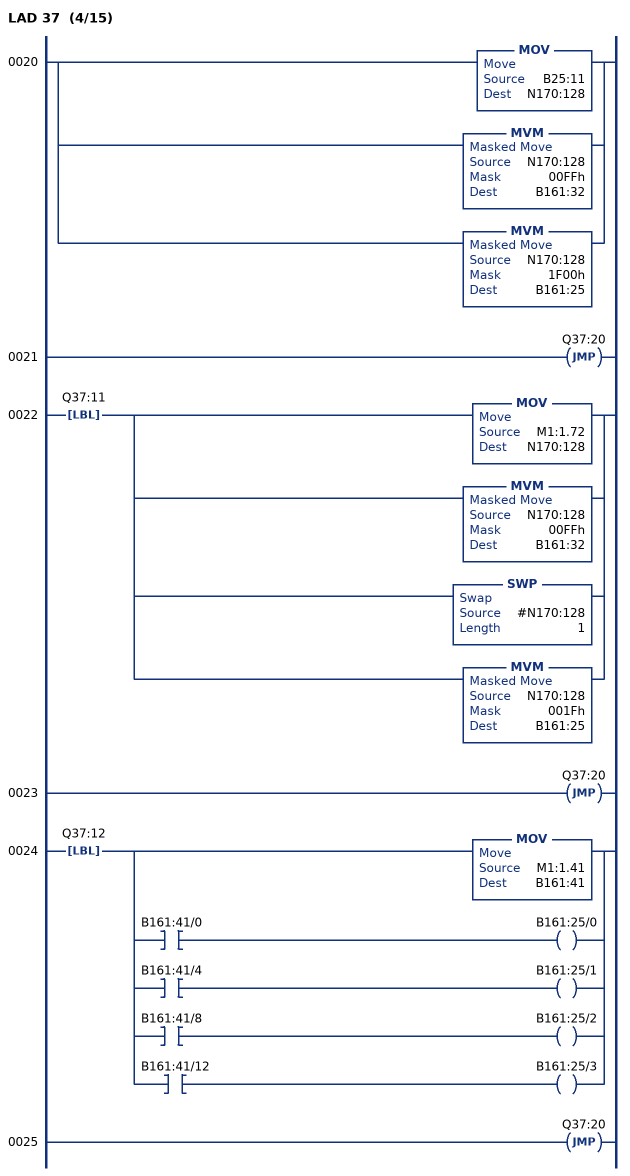
% Rung: 20 %
SOR BST MOV B25:11 N170:128 NXB MVM N170:128 00FFh B161:32 NXB MVM N170:128 1F00h B161:25 BND EOR
% Rung: 21 %
SOR JMP Q37:20 EOR
% Rung: 22 %
SOR LBL Q37:11 BST MOV M1:1.72 N170:128 NXB MVM N170:128 00FFh B161:32 NXB SWP #N170:128 1 NXB MVM N170:128 001Fh B161:25 BND EOR
% Rung: 23 %
SOR JMP Q37:20 EOR
% Rung: 24 %
SOR LBL Q37:12 BST MOV M1:1.41 B161:41 NXB XIC B161:41/0 OTE B161:25/0 NXB XIC B161:41/4 OTE B161:25/1 NXB XIC B161:41/8 OTE B161:25/2 NXB XIC B161:41/12 OTE B161:25/3 BND EOR
% Rung: 25 %
SOR JMP Q37:20 EOR

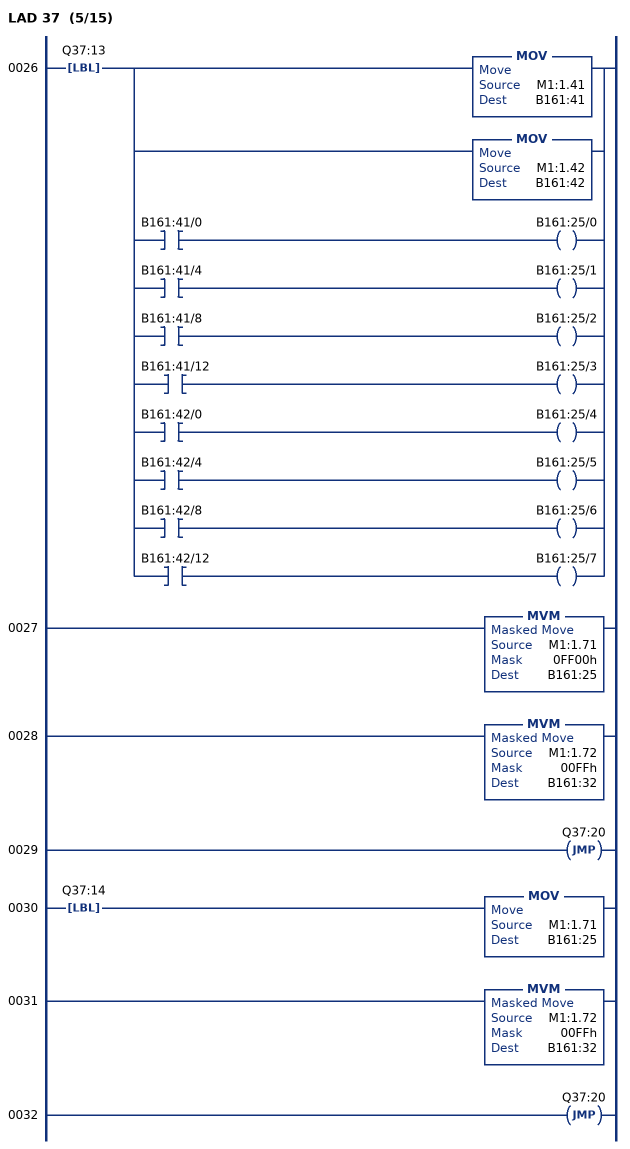
% Rung: 26 %
SOR LBL Q37:13 BST MOV M1:1.41 B161:41 NXB MOV M1:1.42 B161:42 NXB XIC B161:41/0 OTE B161:25/0 NXB XIC B161:41/4 OTE B161:25/1 NXB XIC B161:41/8 OTE B161:25/2 NXB XIC B161:41/12 OTE B161:25/3 NXB XIC B161:42/0 OTE B161:25/4 NXB XIC B161:42/4 OTE B161:25/5 NXB XIC B161:42/8 OTE B161:25/6 NXB XIC B161:42/12 OTE B161:25/7 BND EOR
% Rung: 27 %
SOR MVM M1:1.71 0FF00h B161:25 EOR
% Rung: 28 %
SOR MVM M1:1.72 00FFh B161:32 EOR
% Rung: 29 %
SOR JMP Q37:20 EOR
% Rung: 30 %
SOR LBL Q37:14 MOV M1:1.71 B161:25 EOR
% Rung: 31 %
SOR MVM M1:1.72 00FFh B161:32 EOR
% Rung: 32 %
SOR JMP Q37:20 EOR

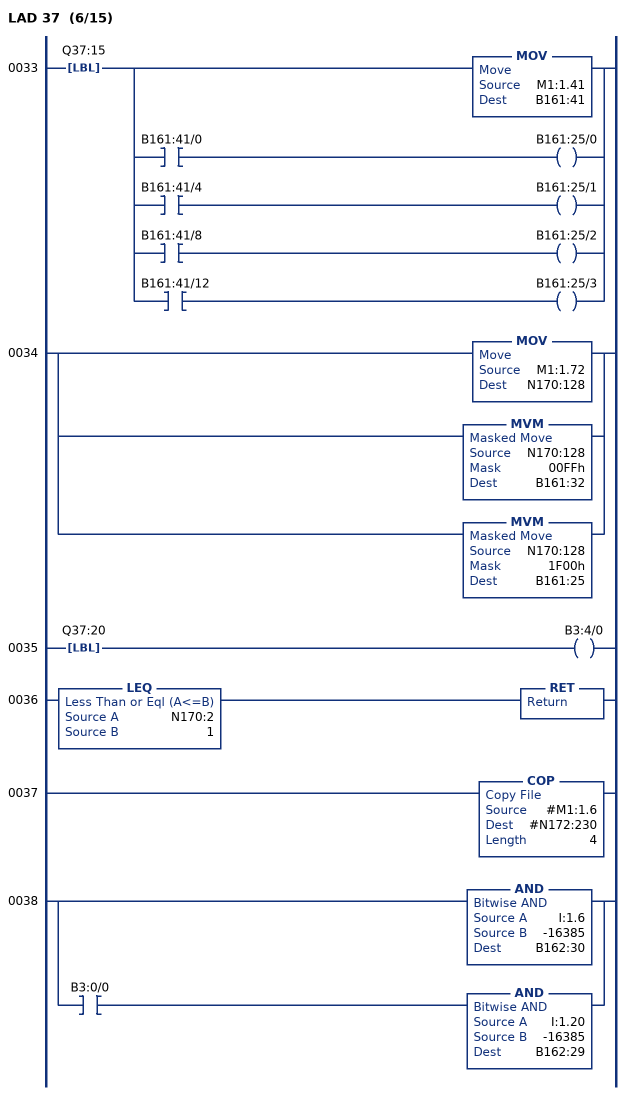
% Rung: 33 %
SOR LBL Q37:15 BST MOV M1:1.41 B161:41 NXB XIC B161:41/0 OTE B161:25/0 NXB XIC B161:41/4 OTE B161:25/1 NXB XIC B161:41/8 OTE B161:25/2 NXB XIC B161:41/12 OTE B161:25/3 BND EOR
% Rung: 34 %
SOR BST MOV M1:1.72 N170:128 NXB MVM N170:128 00FFh B161:32 NXB MVM N170:128 1F00h B161:25 BND EOR
% Rung: 35 %
SOR LBL Q37:20 OTE B3:4/0 EOR
% Rung: 36 %
SOR LEQ N170:2 1 RET EOR
% Rung: 37 %
SOR COP #M1:1.6 #N172:230 4 EOR
% Rung: 38 %
SOR BST AND I:1.6 -16385 B162:30 NXB XIC B3:0/0 AND I:1.20 -16385 B162:29 BND EOR

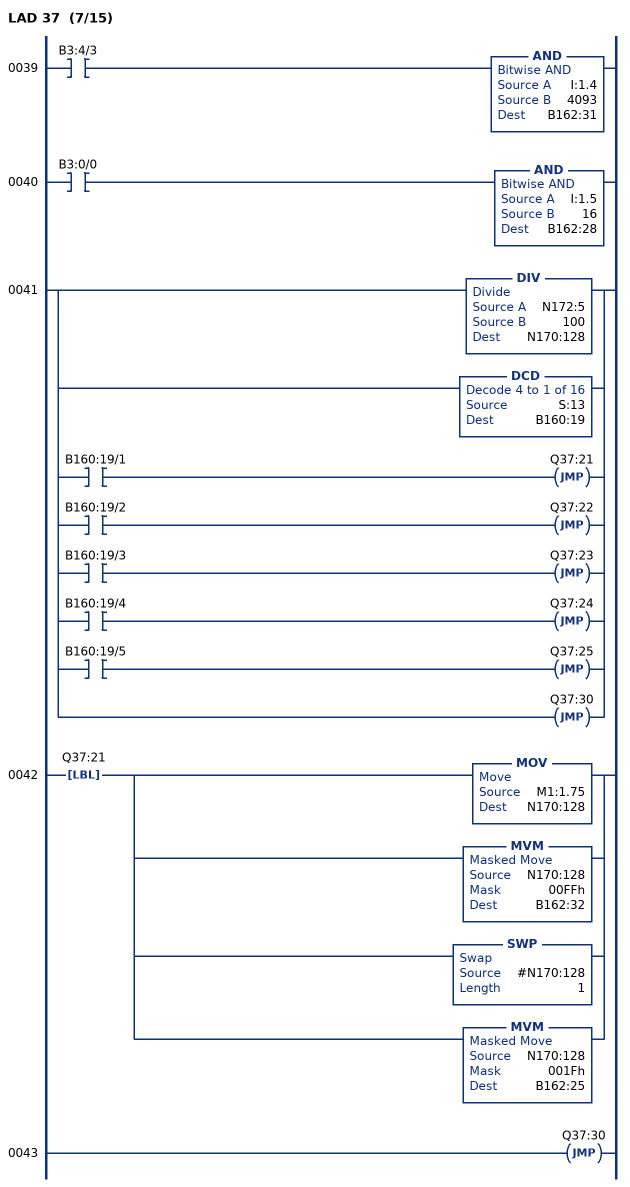
% Rung: 39 %
SOR XIC B3:4/3 AND I:1.4 4093 B162:31 EOR
% Rung: 40 %
SOR XIC B3:0/0 AND I:1.5 16 B162:28 EOR
% Rung: 41 %
SOR BST DIV N172:5 100 N170:128 NXB DCD S:13 B160:19 NXB BST XIC B160:19/1 JMP Q37:21 NXB XIC B160:19/2 JMP Q37:22 NXB XIC B160:19/3 JMP Q37:23 NXB XIC B160:19/4 JMP Q37:24 NXB XIC B160:19/5 JMP Q37:25 BND NXB JMP Q37:30 BND EOR
%   S:13  "Math Register" %
% Rung: 42 %
SOR LBL Q37:21 BST MOV M1:1.75 N170:128 NXB MVM N170:128 00FFh B162:32 NXB SWP #N170:128 1 NXB MVM N170:128 001Fh B162:25 BND EOR
% Rung: 43 %
SOR JMP Q37:30 EOR

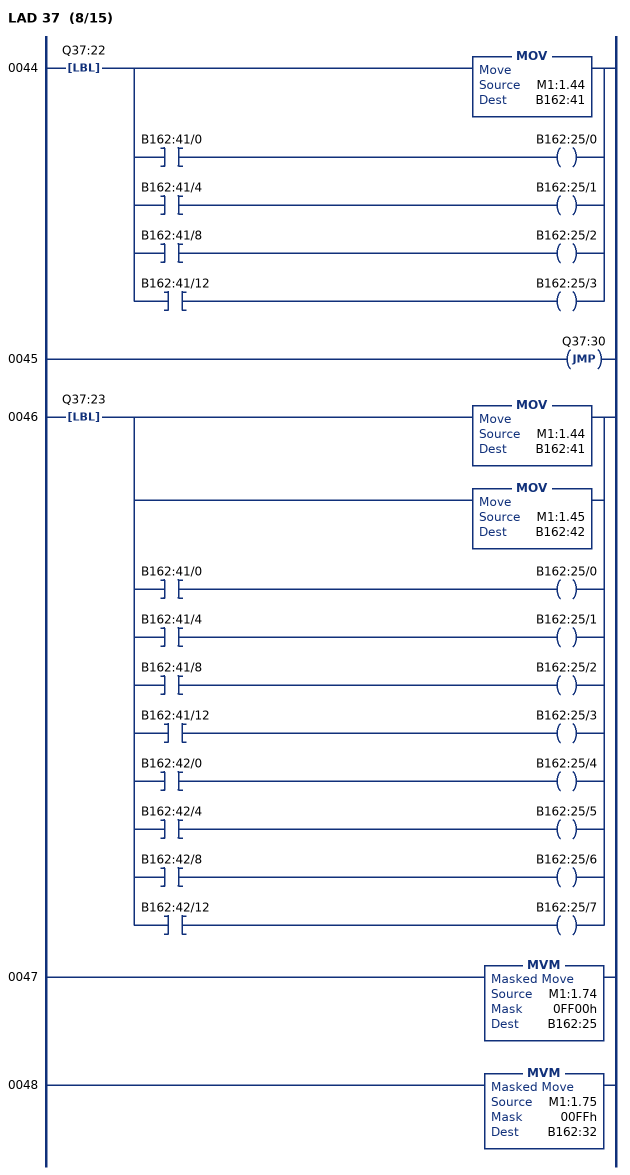
% Rung: 44 %
SOR LBL Q37:22 BST MOV M1:1.44 B162:41 NXB XIC B162:41/0 OTE B162:25/0 NXB XIC B162:41/4 OTE B162:25/1 NXB XIC B162:41/8 OTE B162:25/2 NXB XIC B162:41/12 OTE B162:25/3 BND EOR
% Rung: 45 %
SOR JMP Q37:30 EOR
% Rung: 46 %
SOR LBL Q37:23 BST MOV M1:1.44 B162:41 NXB MOV M1:1.45 B162:42 NXB XIC B162:41/0 OTE B162:25/0 NXB XIC B162:41/4 OTE B162:25/1 NXB XIC B162:41/8 OTE B162:25/2 NXB XIC B162:41/12 OTE B162:25/3 NXB XIC B162:42/0 OTE B162:25/4 NXB XIC B162:42/4 OTE B162:25/5 NXB XIC B162:42/8 OTE B162:25/6 NXB XIC B162:42/12 OTE B162:25/7 BND EOR
% Rung: 47 %
SOR MVM M1:1.74 0FF00h B162:25 EOR
% Rung: 48 %
SOR MVM M1:1.75 00FFh B162:32 EOR

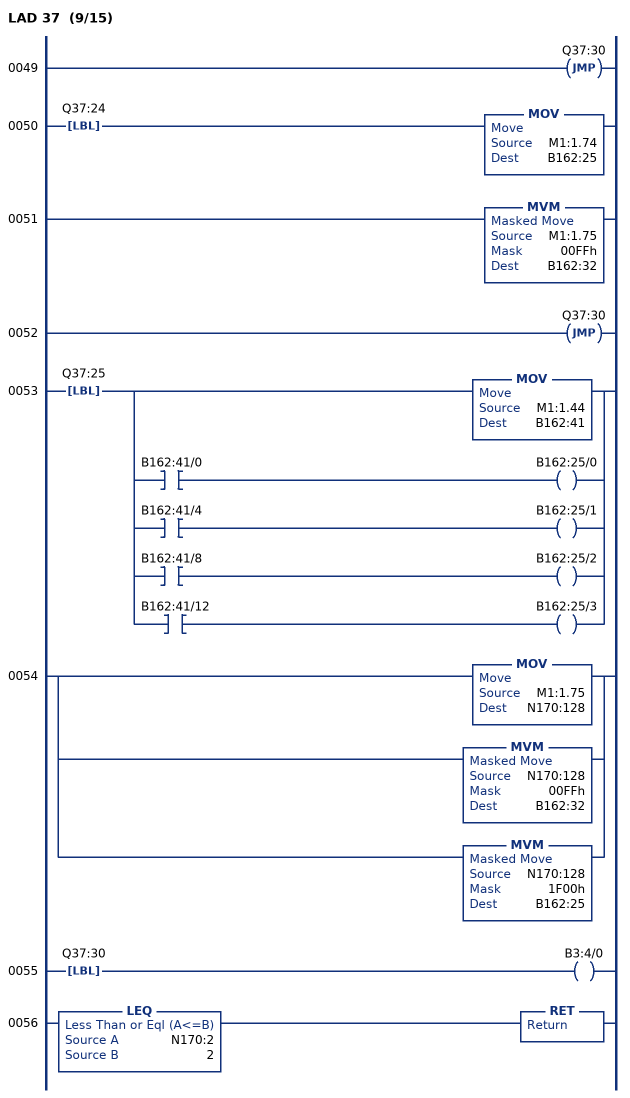
% Rung: 49 %
SOR JMP Q37:30 EOR
% Rung: 50 %
SOR LBL Q37:24 MOV M1:1.74 B162:25 EOR
% Rung: 51 %
SOR MVM M1:1.75 00FFh B162:32 EOR
% Rung: 52 %
SOR JMP Q37:30 EOR
% Rung: 53 %
SOR LBL Q37:25 BST MOV M1:1.44 B162:41 NXB XIC B162:41/0 OTE B162:25/0 NXB XIC B162:41/4 OTE B162:25/1 NXB XIC B162:41/8 OTE B162:25/2 NXB XIC B162:41/12 OTE B162:25/3 BND EOR
% Rung: 54 %
SOR BST MOV M1:1.75 N170:128 NXB MVM N170:128 00FFh B162:32 NXB MVM N170:128 1F00h B162:25 BND EOR
% Rung: 55 %
SOR LBL Q37:30 OTE B3:4/0 EOR
% Rung: 56 %
SOR LEQ N170:2 2 RET EOR

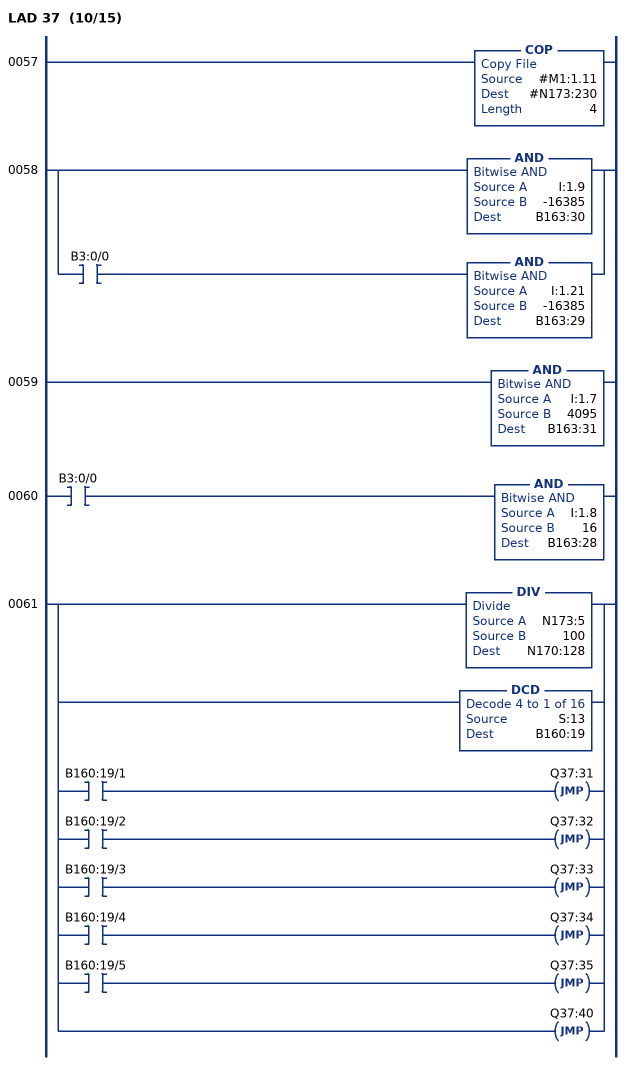
% Rung: 57 %
SOR COP #M1:1.11 #N173:230 4 EOR
% Rung: 58 %
SOR BST AND I:1.9 -16385 B163:30 NXB XIC B3:0/0 AND I:1.21 -16385 B163:29 BND EOR
% Rung: 59 %
SOR AND I:1.7 4095 B163:31 EOR
% Rung: 60 %
SOR XIC B3:0/0 AND I:1.8 16 B163:28 EOR
% Rung: 61 %
SOR BST DIV N173:5 100 N170:128 NXB DCD S:13 B160:19 NXB BST XIC B160:19/1 JMP Q37:31 NXB XIC B160:19/2 JMP Q37:32 NXB XIC B160:19/3 JMP Q37:33 NXB XIC B160:19/4 JMP Q37:34 NXB XIC B160:19/5 JMP Q37:35 BND NXB JMP Q37:40 BND EOR
%   S:13  "Math Register" %

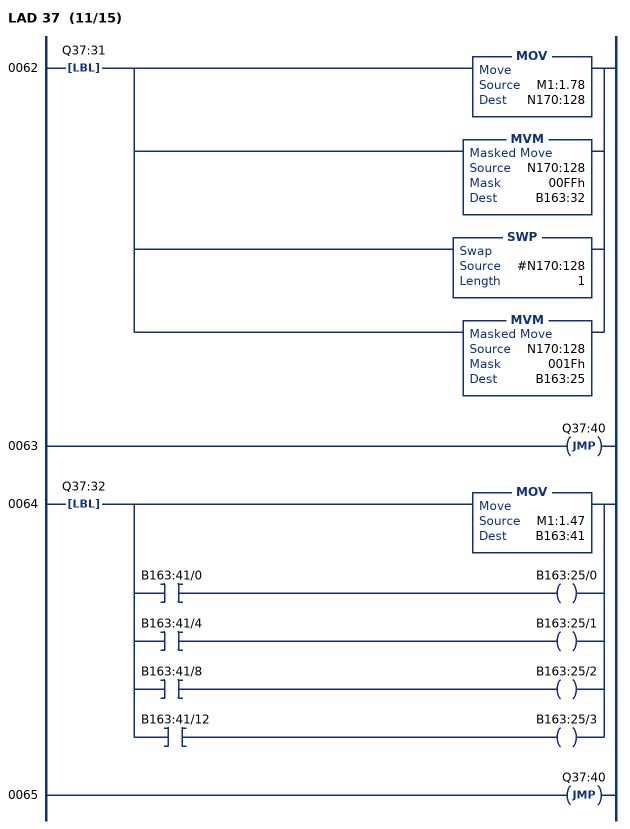
% Rung: 62 %
SOR LBL Q37:31 BST MOV M1:1.78 N170:128 NXB MVM N170:128 00FFh B163:32 NXB SWP #N170:128 1 NXB MVM N170:128 001Fh B163:25 BND EOR
% Rung: 63 %
SOR JMP Q37:40 EOR
% Rung: 64 %
SOR LBL Q37:32 BST MOV M1:1.47 B163:41 NXB XIC B163:41/0 OTE B163:25/0 NXB XIC B163:41/4 OTE B163:25/1 NXB XIC B163:41/8 OTE B163:25/2 NXB XIC B163:41/12 OTE B163:25/3 BND EOR
% Rung: 65 %
SOR JMP Q37:40 EOR

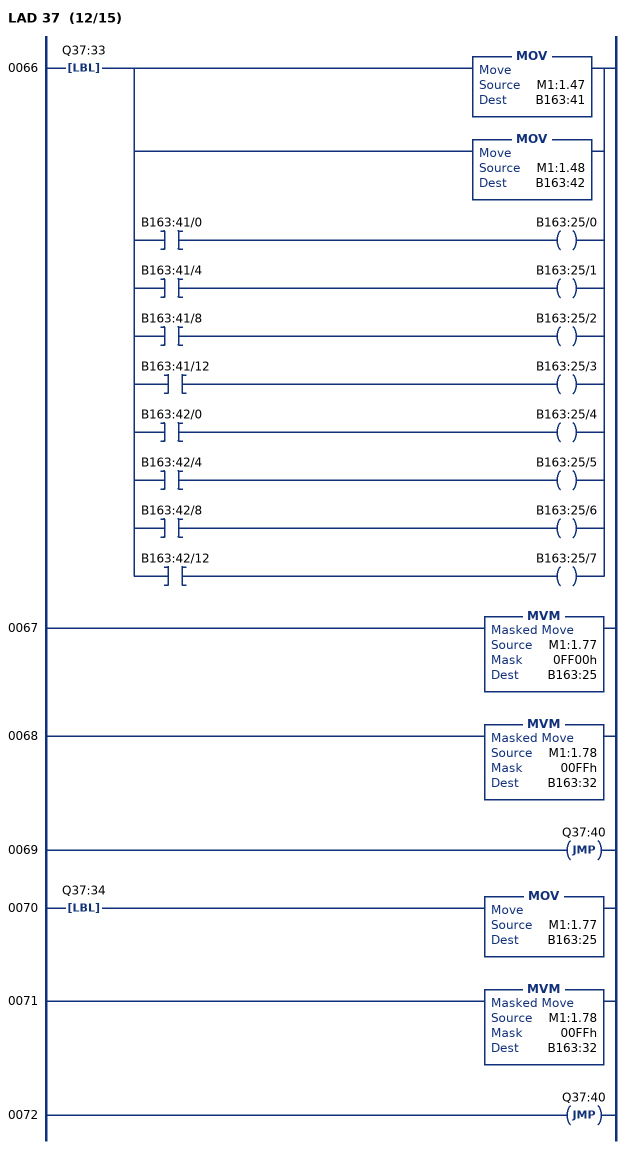
% Rung: 66 %
SOR LBL Q37:33 BST MOV M1:1.47 B163:41 NXB MOV M1:1.48 B163:42 NXB XIC B163:41/0 OTE B163:25/0 NXB XIC B163:41/4 OTE B163:25/1 NXB XIC B163:41/8 OTE B163:25/2 NXB XIC B163:41/12 OTE B163:25/3 NXB XIC B163:42/0 OTE B163:25/4 NXB XIC B163:42/4 OTE B163:25/5 NXB XIC B163:42/8 OTE B163:25/6 NXB XIC B163:42/12 OTE B163:25/7 BND EOR
% Rung: 67 %
SOR MVM M1:1.77 0FF00h B163:25 EOR
% Rung: 68 %
SOR MVM M1:1.78 00FFh B163:32 EOR
% Rung: 69 %
SOR JMP Q37:40 EOR
% Rung: 70 %
SOR LBL Q37:34 MOV M1:1.77 B163:25 EOR
% Rung: 71 %
SOR MVM M1:1.78 00FFh B163:32 EOR
% Rung: 72 %
SOR JMP Q37:40 EOR

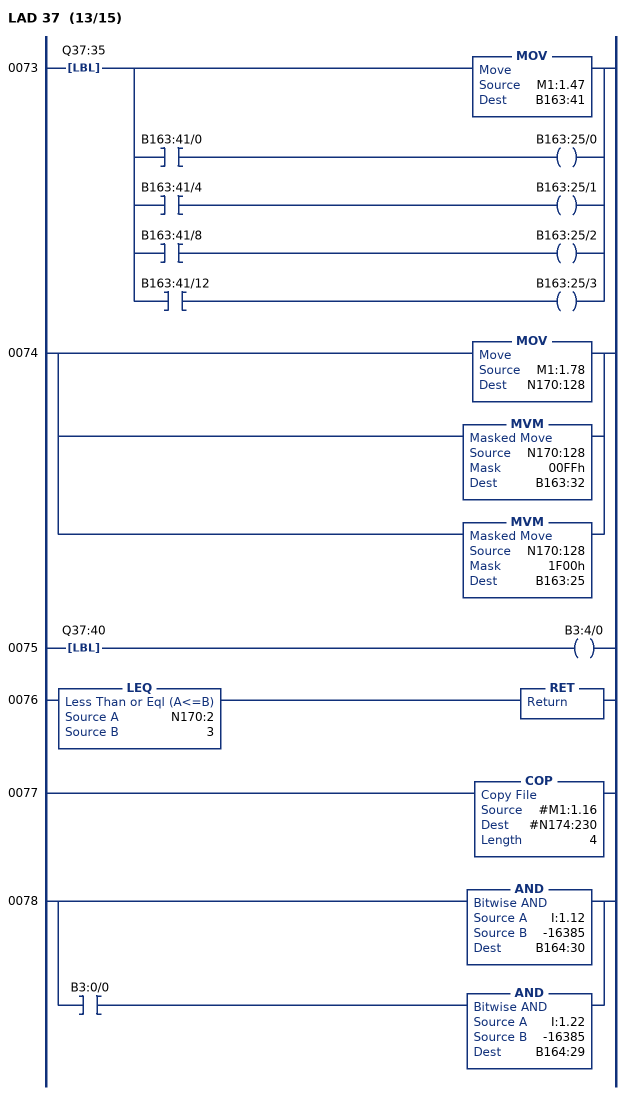
% Rung: 73 %
SOR LBL Q37:35 BST MOV M1:1.47 B163:41 NXB XIC B163:41/0 OTE B163:25/0 NXB XIC B163:41/4 OTE B163:25/1 NXB XIC B163:41/8 OTE B163:25/2 NXB XIC B163:41/12 OTE B163:25/3 BND EOR
% Rung: 74 %
SOR BST MOV M1:1.78 N170:128 NXB MVM N170:128 00FFh B163:32 NXB MVM N170:128 1F00h B163:25 BND EOR
% Rung: 75 %
SOR LBL Q37:40 OTE B3:4/0 EOR
% Rung: 76 %
SOR LEQ N170:2 3 RET EOR
% Rung: 77 %
SOR COP #M1:1.16 #N174:230 4 EOR
% Rung: 78 %
SOR BST AND I:1.12 -16385 B164:30 NXB XIC B3:0/0 AND I:1.22 -16385 B164:29 BND EOR

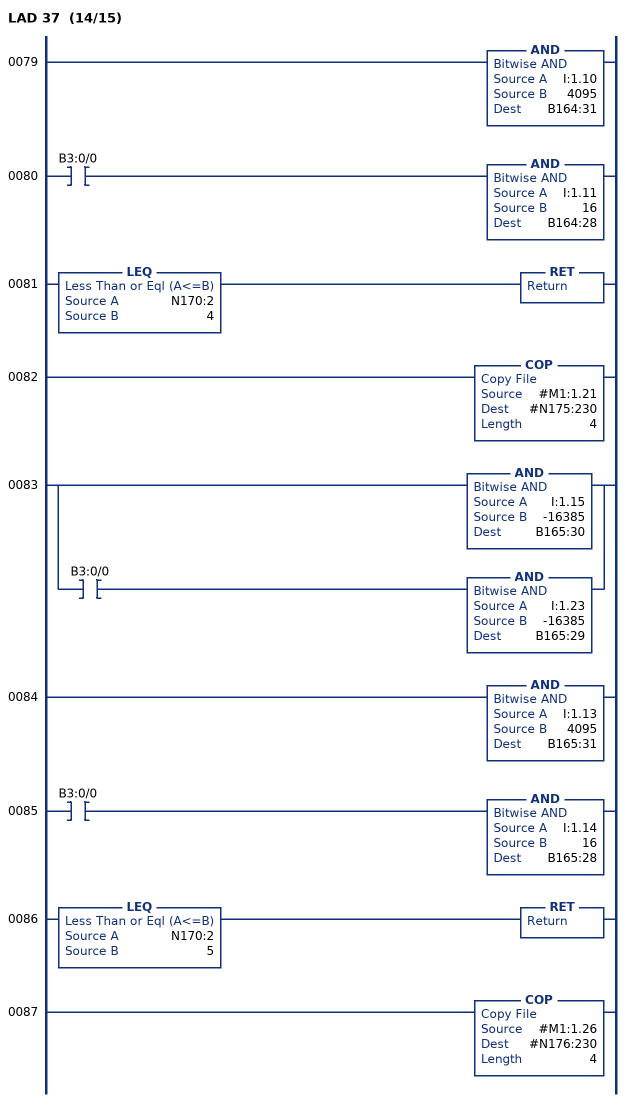
% Rung: 79 %
SOR AND I:1.10 4095 B164:31 EOR
% Rung: 80 %
SOR XIC B3:0/0 AND I:1.11 16 B164:28 EOR
% Rung: 81 %
SOR LEQ N170:2 4 RET EOR
% Rung: 82 %
SOR COP #M1:1.21 #N175:230 4 EOR
% Rung: 83 %
SOR BST AND I:1.15 -16385 B165:30 NXB XIC B3:0/0 AND I:1.23 -16385 B165:29 BND EOR
% Rung: 84 %
SOR AND I:1.13 4095 B165:31 EOR
% Rung: 85 %
SOR XIC B3:0/0 AND I:1.14 16 B165:28 EOR
% Rung: 86 %
SOR LEQ N170:2 5 RET EOR
% Rung: 87 %
SOR COP #M1:1.26 #N176:230 4 EOR

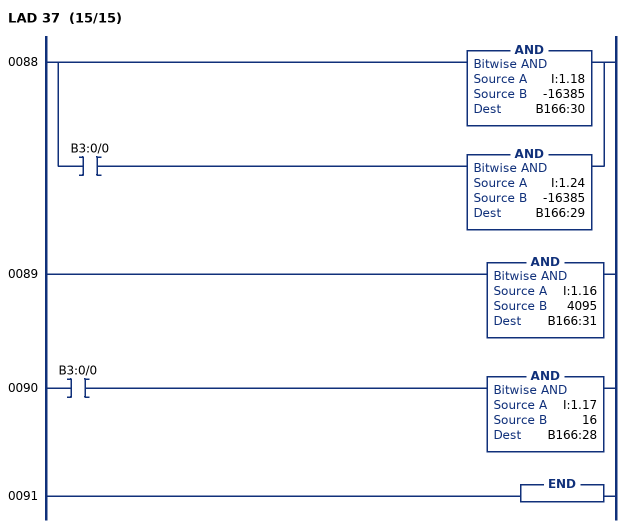
% Rung: 88 %
SOR BST AND I:1.18 -16385 B166:30 NXB XIC B3:0/0 AND I:1.24 -16385 B166:29 BND EOR
% Rung: 89 %
SOR AND I:1.16 4095 B166:31 EOR
% Rung: 90 %
SOR XIC B3:0/0 AND I:1.17 16 B166:28 EOR
% Rung: 91 %
SOR END EOR

LADDER 38
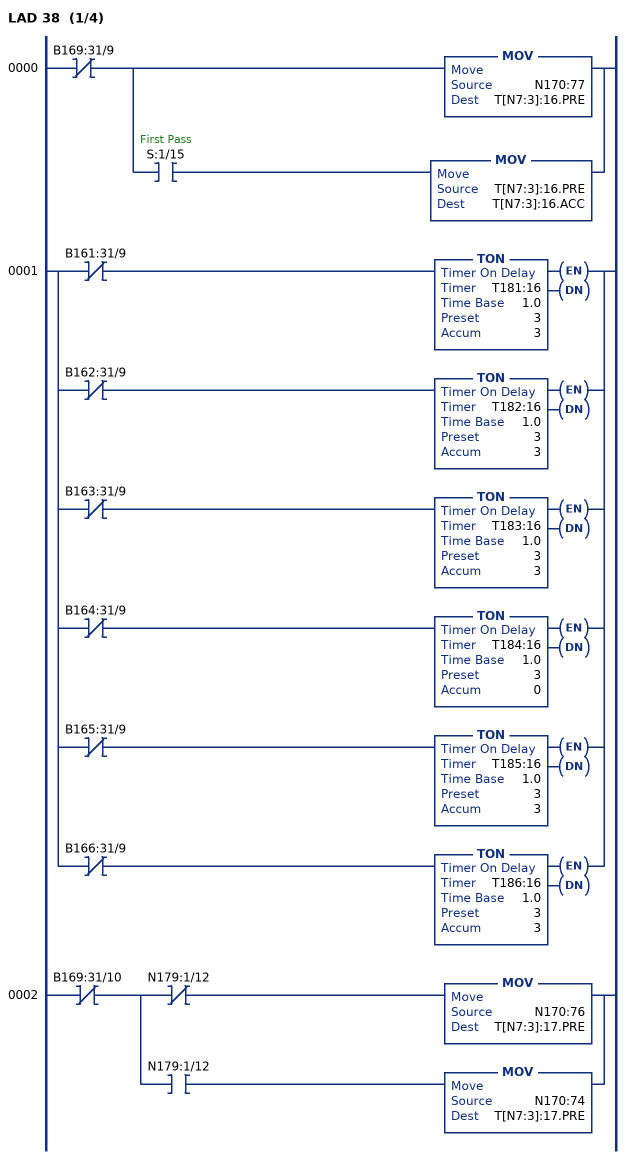
% Rung: 0 %
SOR XIO B169:31/9 BST MOV N170:77 T[N7:3]:16.PRE NXB XIC S:1/15 MOV T[N7:3]:16.PRE T[N7:3]:16.ACC BND EOR
%   S:1/15  "First Pass" %
% Rung: 1 %
SOR BST XIO B161:31/9 TON T181:16 1.0 3 3 NXB XIO B162:31/9 TON T182:16 1.0 3 3 NXB XIO B163:31/9 TON T183:16 1.0 3 3 NXB XIO B164:31/9 TON T184:16 1.0 3 0 NXB XIO B165:31/9 TON T185:16 1.0 3 3 NXB XIO B166:31/9 TON T186:16 1.0 3 3 BND EOR
% Rung: 2 %
SOR XIO B169:31/10 BST XIO N179:1/12 MOV N170:76 T[N7:3]:17.PRE NXB XIC N179:1/12 MOV N170:74 T[N7:3]:17.PRE BND EOR

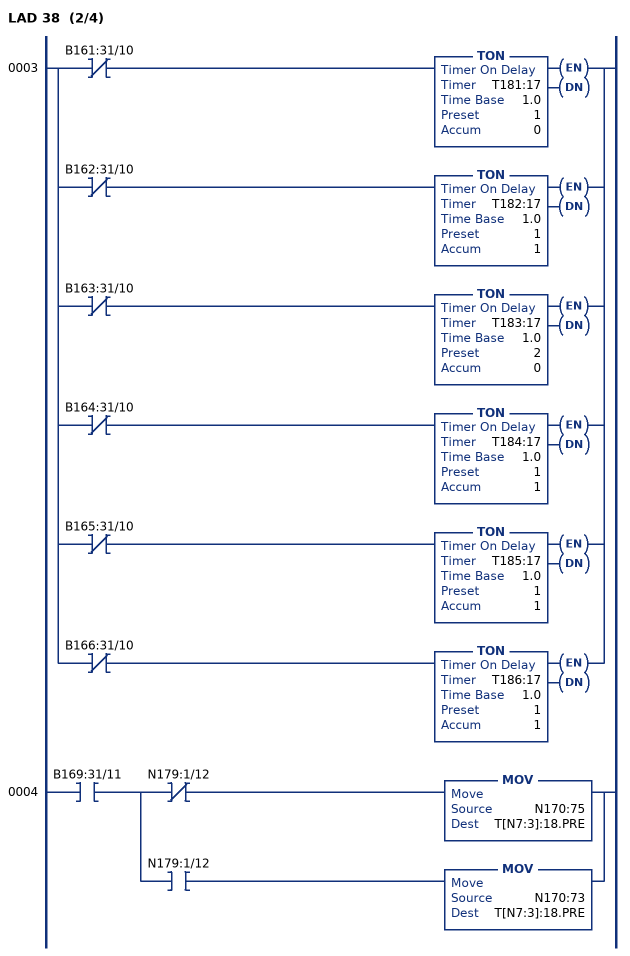
% Rung: 3 %
SOR BST XIO B161:31/10 TON T181:17 1.0 1 0 NXB XIO B162:31/10 TON T182:17 1.0 1 1 NXB XIO B163:31/10 TON T183:17 1.0 2 0 NXB XIO B164:31/10 TON T184:17 1.0 1 1 NXB XIO B165:31/10 TON T185:17 1.0 1 1 NXB XIO B166:31/10 TON T186:17 1.0 1 1 BND EOR
% Rung: 4 %
SOR XIC B169:31/11 BST XIO N179:1/12 MOV N170:75 T[N7:3]:18.PRE NXB XIC N179:1/12 MOV N170:73 T[N7:3]:18.PRE BND EOR

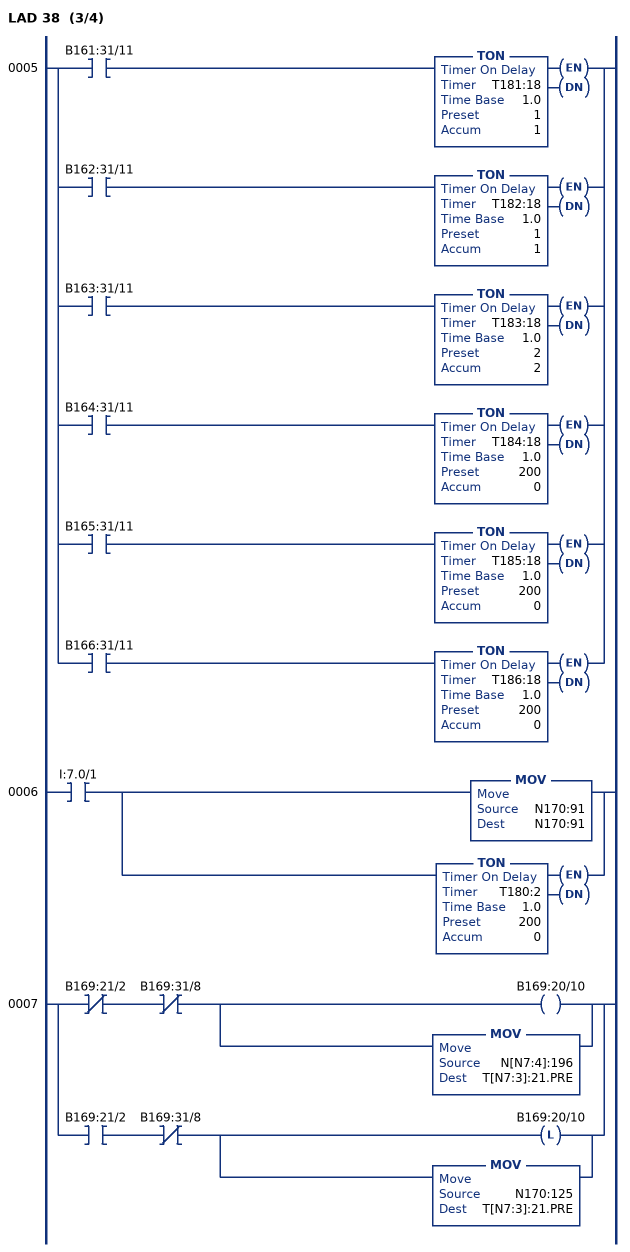
% Rung: 5 %
SOR BST XIC B161:31/11 TON T181:18 1.0 1 1 NXB XIC B162:31/11 TON T182:18 1.0 1 1 NXB XIC B163:31/11 TON T183:18 1.0 2 2 NXB XIC B164:31/11 TON T184:18 1.0 200 0 NXB XIC B165:31/11 TON T185:18 1.0 200 0 NXB XIC B166:31/11 TON T186:18 1.0 200 0 BND EOR
% Rung: 6 %
SOR XIC I:7.0/1 BST MOV N170:91 N170:91 NXB TON T180:2 1.0 200 0 BND EOR
% Rung: 7 %
SOR BST XIO B169:21/2 XIO B169:31/8 BST OTE B169:20/10 NXB MOV N[N7:4]:196 T[N7:3]:21.PRE BND NXB XIC B169:21/2 XIO B169:31/8 BST OTL B169:20/10 NXB MOV N170:125 T[N7:3]:21.PRE BND BND EOR

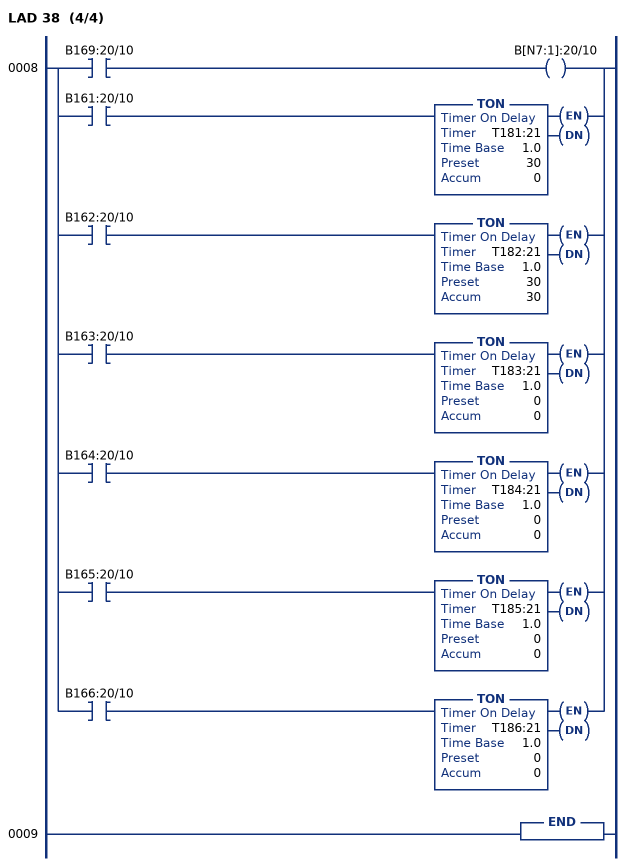
% Rung: 8 %
SOR BST XIC B169:20/10 OTE B[N7:1]:20/10 NXB XIC B161:20/10 TON T181:21 1.0 30 0 NXB XIC B162:20/10 TON T182:21 1.0 30 30 NXB XIC B163:20/10 TON T183:21 1.0 0 0 NXB XIC B164:20/10 TON T184:21 1.0 0 0 NXB XIC B165:20/10 TON T185:21 1.0 0 0 NXB XIC B166:20/10 TON T186:21 1.0 0 0 BND EOR
% Rung: 9 %
SOR END EOR

LADDER 39
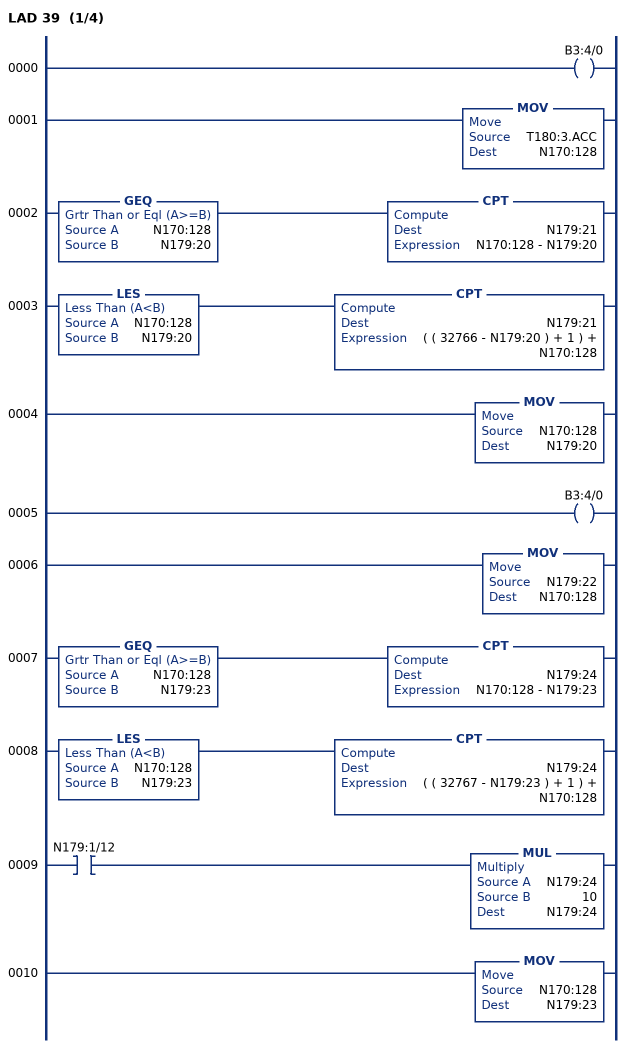
% Rung: 0 %
SOR OTE B3:4/0 EOR
% Rung: 1 %
SOR MOV T180:3.ACC N170:128 EOR
% Rung: 2 %
SOR GEQ N170:128 N179:20 CPT N179:21 " N170:128 - N179:20 " EOR
% Rung: 3 %
SOR LES N170:128 N179:20 CPT N179:21 " ( ( 32766 - N179:20 ) + 1 ) + N170:128 " EOR
% Rung: 4 %
SOR MOV N170:128 N179:20 EOR
% Rung: 5 %
SOR OTE B3:4/0 EOR
% Rung: 6 %
SOR MOV N179:22 N170:128 EOR
% Rung: 7 %
SOR GEQ N170:128 N179:23 CPT N179:24 " N170:128 - N179:23 " EOR
% Rung: 8 %
SOR LES N170:128 N179:23 CPT N179:24 " ( ( 32767 - N179:23 ) + 1 ) + N170:128 " EOR
% Rung: 9 %
SOR XIC N179:1/12 MUL N179:24 10 N179:24 EOR
% Rung: 10 %
SOR MOV N170:128 N179:23 EOR

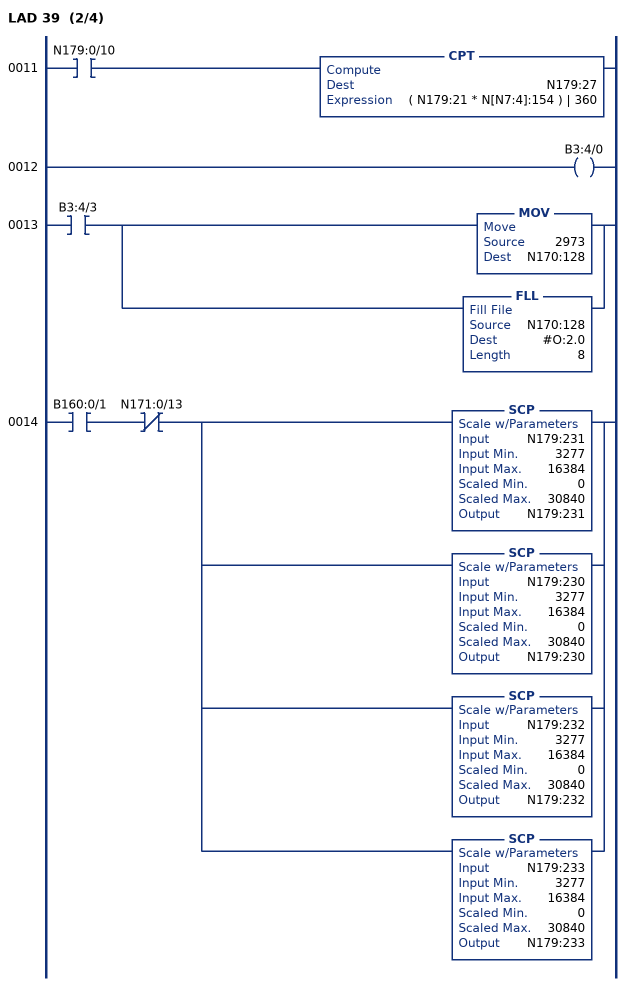
% Rung: 11 %
SOR XIC N179:0/10 CPT N179:27 " ( N179:21 * N[N7:4]:154 ) | 360 " EOR
% Rung: 12 %
SOR OTE B3:4/0 EOR
% Rung: 13 %
SOR XIC B3:4/3 BST MOV 2973 N170:128 NXB FLL N170:128 #O:2.0 8 BND EOR
% Rung: 14 %
SOR XIC B160:0/1 XIO N171:0/13 BST SCP N179:231 3277 16384 0 30840 N179:231 NXB SCP N179:230 3277 16384 0 30840 N179:230 NXB SCP N179:232 3277 16384 0 30840 N179:232 NXB SCP N179:233 3277 16384 0 30840 N179:233 BND EOR

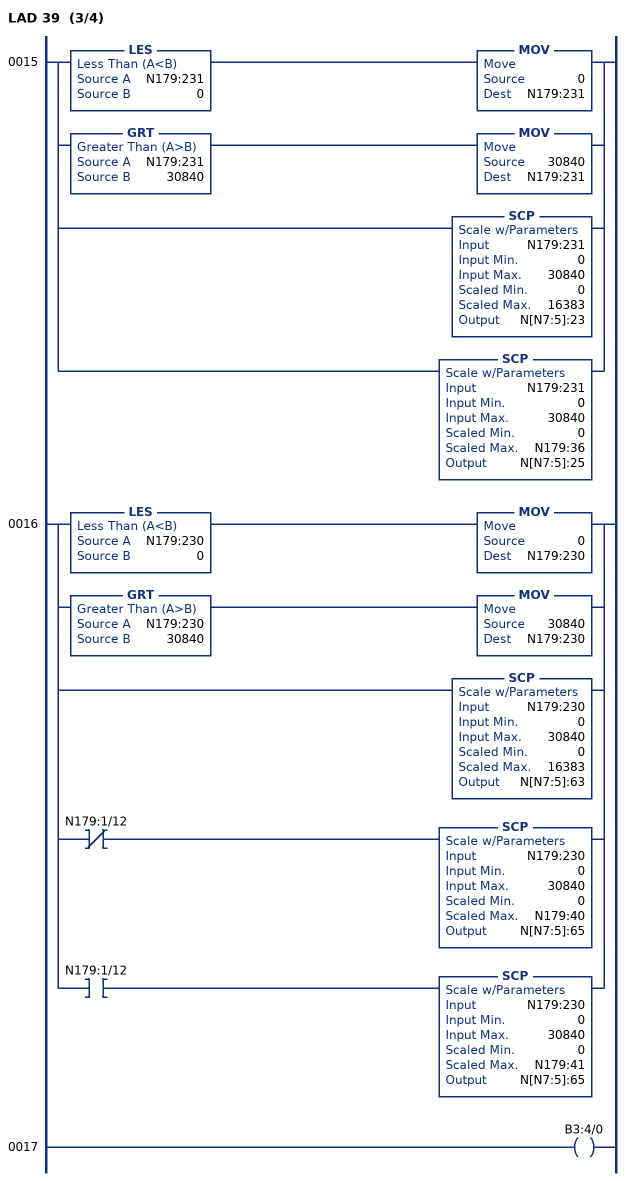
% Rung: 15 %
SOR BST LES N179:231 0 MOV 0 N179:231 NXB GRT N179:231 30840 MOV 30840 N179:231 NXB SCP N179:231 0 30840 0 16383 N[N7:5]:23 NXB SCP N179:231 0 30840 0 N179:36 N[N7:5]:25 BND EOR
% Rung: 16 %
SOR BST LES N179:230 0 MOV 0 N179:230 NXB GRT N179:230 30840 MOV 30840 N179:230 NXB SCP N179:230 0 30840 0 16383 N[N7:5]:63 NXB XIO N179:1/12 SCP N179:230 0 30840 0 N179:40 N[N7:5]:65 NXB XIC N179:1/12 SCP N179:230 0 30840 0 N179:41 N[N7:5]:65 BND EOR
% Rung: 17 %
SOR OTE B3:4/0 EOR

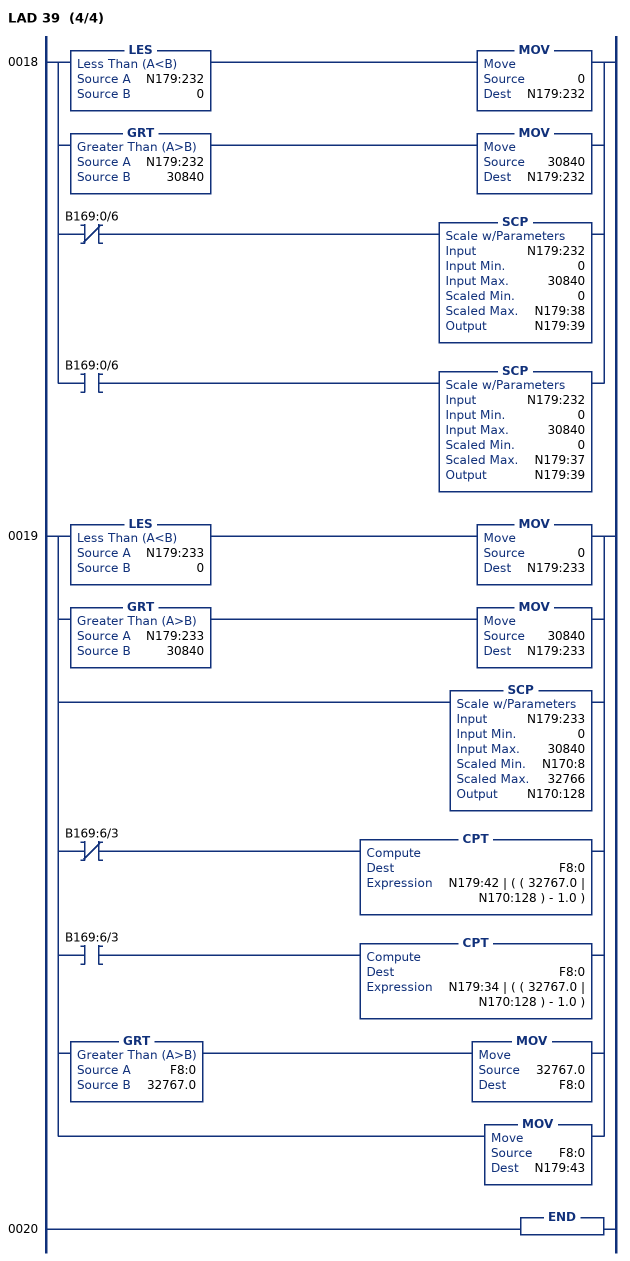
% Rung: 18 %
SOR BST LES N179:232 0 MOV 0 N179:232 NXB GRT N179:232 30840 MOV 30840 N179:232 NXB XIO B169:0/6 SCP N179:232 0 30840 0 N179:38 N179:39 NXB XIC B169:0/6 SCP N179:232 0 30840 0 N179:37 N179:39 BND EOR
% Rung: 19 %
SOR BST LES N179:233 0 MOV 0 N179:233 NXB GRT N179:233 30840 MOV 30840 N179:233 NXB SCP N179:233 0 30840 N170:8 32766 N170:128 NXB BST XIO B169:6/3 CPT F8:0 " N179:42 | ( ( 32767.0 | N170:128 ) - 1.0 ) " NXB XIC B169:6/3 CPT F8:0 " N179:34 | ( ( 32767.0 | N170:128 ) - 1.0 ) " BND NXB GRT F8:0 32767.0 MOV 32767.0 F8:0 NXB MOV F8:0 N179:43 BND EOR
% Rung: 20 %
SOR END EOR

LADDER 40
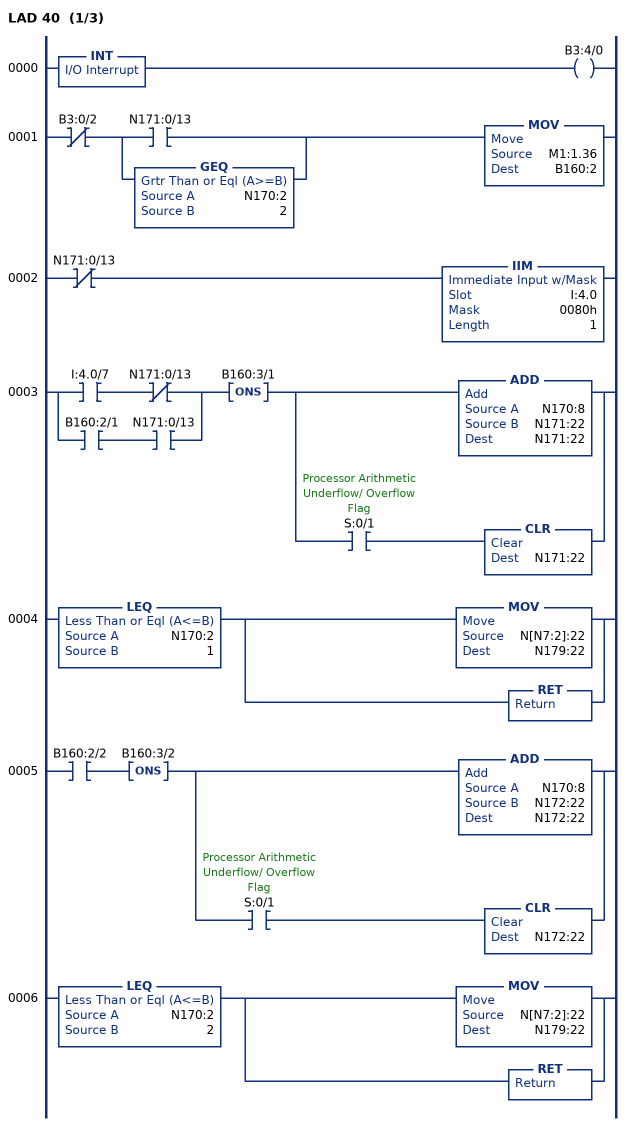
% Rung: 0 %
SOR INT OTE B3:4/0 EOR
% Rung: 1 %
SOR XIO B3:0/2 BST XIC N171:0/13 NXB GEQ N170:2 2 BND MOV M1:1.36 B160:2 EOR
% Rung: 2 %
SOR XIO N171:0/13 IIM I:4.0 0080h 1 EOR
% Rung: 3 %
SOR BST XIC I:4.0/7 XIO N171:0/13 NXB XIC B160:2/1 XIC N171:0/13 BND OSR B160:3/1 BST ADD N170:8 N171:22 N171:22 NXB XIC S:0/1 CLR N171:22 BND EOR
%   S:0/1  "Processor Arithmetic Underflow/ Overflow Flag" %
% Rung: 4 %
SOR LEQ N170:2 1 BST MOV N[N7:2]:22 N179:22 NXB RET BND EOR
% Rung: 5 %
SOR XIC B160:2/2 OSR B160:3/2 BST ADD N170:8 N172:22 N172:22 NXB XIC S:0/1 CLR N172:22 BND EOR
%   S:0/1  "Processor Arithmetic Underflow/ Overflow Flag" %
% Rung: 6 %
SOR LEQ N170:2 2 BST MOV N[N7:2]:22 N179:22 NXB RET BND EOR

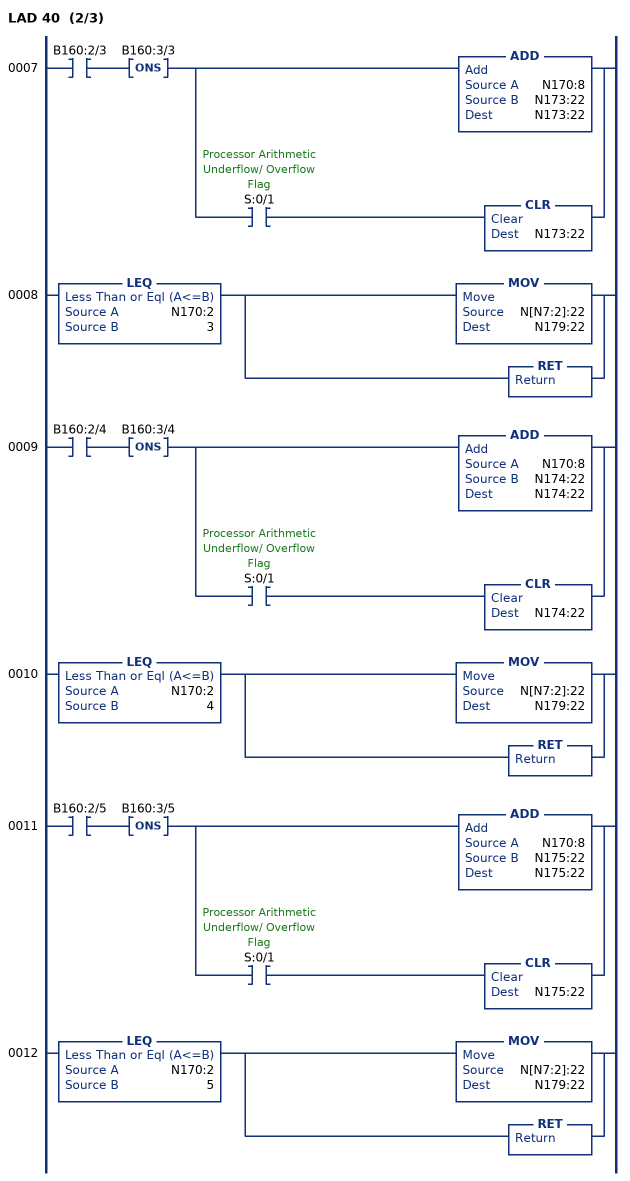
% Rung: 7 %
SOR XIC B160:2/3 OSR B160:3/3 BST ADD N170:8 N173:22 N173:22 NXB XIC S:0/1 CLR N173:22 BND EOR
%   S:0/1  "Processor Arithmetic Underflow/ Overflow Flag" %
% Rung: 8 %
SOR LEQ N170:2 3 BST MOV N[N7:2]:22 N179:22 NXB RET BND EOR
% Rung: 9 %
SOR XIC B160:2/4 OSR B160:3/4 BST ADD N170:8 N174:22 N174:22 NXB XIC S:0/1 CLR N174:22 BND EOR
%   S:0/1  "Processor Arithmetic Underflow/ Overflow Flag" %
% Rung: 10 %
SOR LEQ N170:2 4 BST MOV N[N7:2]:22 N179:22 NXB RET BND EOR
% Rung: 11 %
SOR XIC B160:2/5 OSR B160:3/5 BST ADD N170:8 N175:22 N175:22 NXB XIC S:0/1 CLR N175:22 BND EOR
%   S:0/1  "Processor Arithmetic Underflow/ Overflow Flag" %
% Rung: 12 %
SOR LEQ N170:2 5 BST MOV N[N7:2]:22 N179:22 NXB RET BND EOR

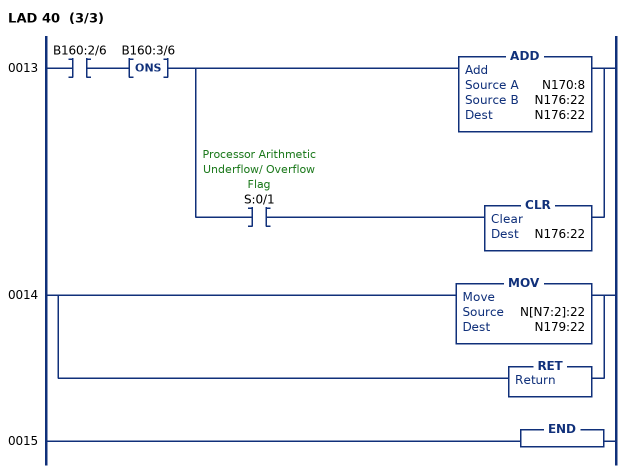
% Rung: 13 %
SOR XIC B160:2/6 OSR B160:3/6 BST ADD N170:8 N176:22 N176:22 NXB XIC S:0/1 CLR N176:22 BND EOR
%   S:0/1  "Processor Arithmetic Underflow/ Overflow Flag" %
% Rung: 14 %
SOR BST MOV N[N7:2]:22 N179:22 NXB RET BND EOR
% Rung: 15 %
SOR END EOR

LADDER 41
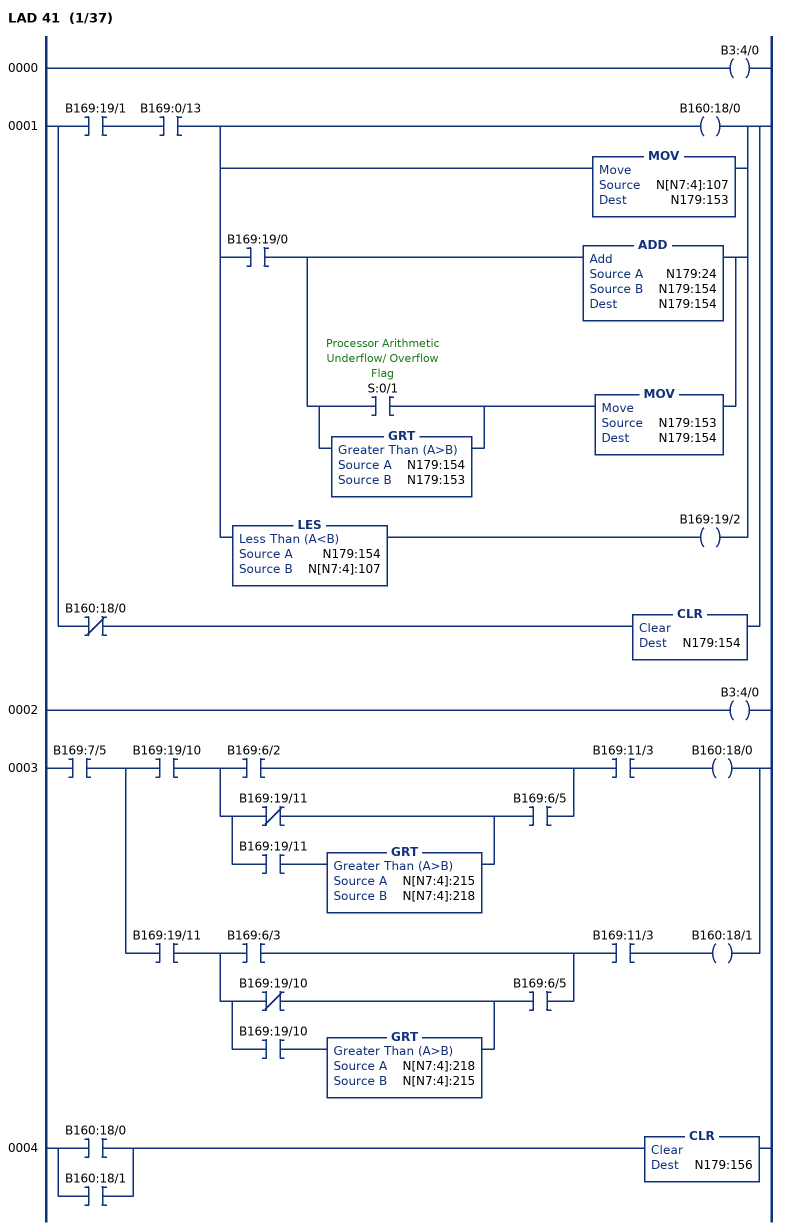
% Rung: 0 %
SOR OTE B3:4/0 EOR
% Rung: 1 %
SOR BST XIC B169:19/1 XIC B169:0/13 BST BST OTE B160:18/0 NXB MOV N[N7:4]:107 N179:153 BND NXB XIC B169:19/0 BST ADD N179:24 N179:154 N179:154 NXB BST XIC S:0/1 NXB GRT N179:154 N179:153 BND MOV N179:153 N179:154 BND NXB LES N179:154 N[N7:4]:107 OTE B169:19/2 BND NXB XIO B160:18/0 CLR N179:154 BND EOR
%   S:0/1  "Processor Arithmetic Underflow/ Overflow Flag" %
% Rung: 2 %
SOR OTE B3:4/0 EOR
% Rung: 3 %
SOR XIC B169:7/5 BST XIC B169:19/10 BST XIC B169:6/2 NXB BST XIO B169:19/11 NXB XIC B169:19/11 GRT N[N7:4]:215 N[N7:4]:218 BND XIC B169:6/5 BND XIC B169:11/3 OTE B160:18/0 NXB XIC B169:19/11 BST XIC B169:6/3 NXB BST XIO B169:19/10 NXB XIC B169:19/10 GRT N[N7:4]:218 N[N7:4]:215 BND XIC B169:6/5 BND XIC B169:11/3 OTE B160:18/1 BND EOR
% Rung: 4 %
SOR BST XIC B160:18/0 NXB XIC B160:18/1 BND CLR N179:156 EOR

